// TIA Portal V15 export
// export: Created 2019-02-11T17:35:24.3452178Z, ExportSetting WithDefaults, WithReadOnly, DisplayName Totally Integrated Automation Portal, DisplayVersion V15 Update 2, DisplayName TIA Portal Openness, DisplayVersion V15 Update 2, DisplayName STEP 7 Professional, DisplayVersion V15 Update 2, DisplayName STEP 7 Safety, DisplayVersion V15, DisplayName WinCC Professional, DisplayVersion V15 Update 2, DisplayName SIMATIC Visualization Architect, DisplayVersion V15 Update 1
DATA_BLOCK "FGDB_ROBNAME@StudWeld"   // DB37
{ S7_Optimized_Access := 'FALSE' }
AUTHOR : integra
FAMILY : SUB
VERSION : 1.0
// stored: AutoNumber true, CodeModifiedDate 2019-02-11T17:32:35.5704024Z, CompileDate 2019-02-11T17:35:11.3679114Z, CreationDate 2019-02-11T17:32:35.4877706Z, DBAccessibleFromOPCUA true, InstanceOfName iSF_TECH_ROBOT_STUD_WELDING, InstanceOfNumber 15, InstanceOfType FB, InterfaceModifiedDate 2019-02-11T17:15:28.4108745Z, IsConsistent true, IsKnowHowProtected false, ModifiedDate 2019-02-11T17:32:35.5704024Z, ParameterModified 2018-10-24T10:12:24.9668345Z, StructureModified 2018-10-24T10:12:24.9668345Z, UDAEnableTagReadback false
"iSF_TECH_ROBOT_STUD_WELDING"
   // VAR_INPUT
   //    fct : Int;
   //    safetyStop : Bool;
   //    functionPoint : String[6];
   //    identType : String[12];
   //    releaseALUwelding : Bool;
   // END_VAR
   // VAR_OUTPUT
   //    qualityDataSent : Bool;
   //    qStop : Bool;
   //    counterParts : Int;
   //    counterNIOpoints : Int;
   //    counterIOpoints : Int;
   //    requestALUwelding : Bool;
   //    headClean1HomePosition : Bool;
   //    headClean2HomePosition : Bool;
   //    headClean3HomePosition : Bool;
   //    fault : Bool;
   // END_VAR
   // VAR_IN_OUT
   //    IfcFGExternal : "iUDT_IFC_SYS_EXTERNAL_ALARM";
   //    IfcTECH : "iUDT_IFC_ROBOT_TECH";
   //    IfcAcyclicdata : "iUDT_IFC_ROBOT_ACYCLICDATA";
   //    ident : Variant;
   //    IfcTLG : "iUDT_IFC_TLG";
   //    TLG_MQDV : "iUDT_TLG_MQDV_ROBOT";
   //    TLG_ENEV : "iUDT_TLG_ENEV";
   //    In_PI_TECH : "iUDT_PI_ROBOT_ADRxx48_TECH";
   //    Out_PO_TECH : "iUDT_PO_ROBOT_ADRxx48_TECH";
   // END_VAR
   // VAR
   //    F : Struct
   //       wrongID : Bool;
   //       notReady : Bool;
   //       boltControllerfault : Bool;
   //       plus : Bool;
   //       pointsNIO : Bool;
   //       partsNIO : Bool;
   //    END_STRUCT;
   //    Masks : Struct
   //       disableFault1_8 : Byte;
   //       prodRelevantFault1_8 : Byte;
   //    END_STRUCT;
   //    LastState : Struct
   //       fault1_8 : Byte;
   //    END_STRUCT;
   //    Tmr : Struct
   //       s1 { S7_SetPoint := 'True'} : Int;
   //       a1 : Int;
   //    END_STRUCT;
   //    TmrB : Struct
   //       "1_EnableDelayTime" : Bool;
   //       "1_RunDelayTime" : Bool;
   //       "1_DoneDelayTime" : Bool;
   //    END_STRUCT;
   //    D : Struct
   //       visuAck : Bool;
   //       evaluatedNIOCounter : Bool;
   //    END_STRUCT;
   //    V : Struct
   //       pointsNIO : Struct
   //          actual : Int;
   //          limitValue { S7_SetPoint := 'True'} : Int;
   //       END_STRUCT;
   //       partsNIO : Struct
   //          actual : Int;
   //          limitValue { S7_SetPoint := 'True'} : Int;
   //          resetCounter { S7_SetPoint := 'True'} : Int;
   //          actualCounter : Int;
   //       END_STRUCT;
   //       plusNIO : Struct
   //          actual : Int;
   //          limitValue { S7_SetPoint := 'True'} : Int;
   //          resetCounter { S7_SetPoint := 'True'} : Int;
   //          actualCounter : Int;
   //       END_STRUCT;
   //    END_STRUCT;
   //    TECH : Struct
   //       ID : Byte;
   //       ready : Bool;
   //       noFault : Bool;
   //       warning : Bool;
   //       noEstop : Bool;
   //       noUserProtection : Bool;
   //       plus : Bool;
   //       tolerance : Bool;
   //       requestALUwelding : Bool;
   //       preWarningHeadClean : Bool;
   //       requestHeadClean : Bool;
   //       headCleanOverflow : Bool;
   //       headCleanRotateSwitch : Bool;
   //       headClean1WorkPosition : Bool;
   //       headClean1HomePosition : Bool;
   //       headClean2WorkPosition : Bool;
   //       headClean2HomePosition : Bool;
   //       headClean3WorkPosition : Bool;
   //       headClean3HomePosition : Bool;
   //       technoBit19 : Bool;
   //       technoBit20 : Bool;
   //       technoBit21 : Bool;
   //       technoBit22 : Bool;
   //       technoBit23 : Bool;
   //       technoBit24 : Bool;
   //       technoBit25 : Bool;
   //       technoBit26 : Bool;
   //       technoBit27 : Bool;
   //       technoBit28 : Bool;
   //       technoBit29 : Bool;
   //       technoBit30 : Bool;
   //       technoBit31 : Bool;
   //       technoBit32 : Bool;
   //       technoBit33 : Bool;
   //       technoBit34 : Bool;
   //       technoBit35 : Bool;
   //       technoBit36 : Bool;
   //       technoBit37 : Bool;
   //       technoBit38 : Bool;
   //       technoBit39 : Bool;
   //       technoBit40 : Bool;
   //    END_STRUCT;
   //    TECH_OUT : Struct
   //       ID { ExternalWritable := 'False'} : Byte;
   //       releaseALUwelding : Bool;
   //       technoBit2 : Bool;
   //       technoBit3 : Bool;
   //       technoBit4 : Bool;
   //       technoBit5 : Bool;
   //       technoBit6 : Bool;
   //       technoBit7 : Bool;
   //       technoBit8 : Bool;
   //       technoBit9 : Bool;
   //       technoBit10 : Bool;
   //       technoBit11 : Bool;
   //       technoBit12 : Bool;
   //       technoBit13 : Bool;
   //       technoBit14 : Bool;
   //       technoBit15 : Bool;
   //       technoBit16 : Bool;
   //       technoBit17 : Bool;
   //       technoBit18 : Bool;
   //       technoBit19 : Bool;
   //       technoBit20 : Bool;
   //       technoBit21 : Bool;
   //       technoBit22 : Bool;
   //       technoBit23 : Bool;
   //       technoBit24 : Bool;
   //       technoBit25 : Bool;
   //       technoBit26 : Bool;
   //       technoBit27 : Bool;
   //       technoBit28 : Bool;
   //       technoBit29 : Bool;
   //       technoBit30 : Bool;
   //       technoBit31 : Bool;
   //       technoBit32 : Bool;
   //       technoBit33 : Bool;
   //       technoBit34 : Bool;
   //       technoBit35 : Bool;
   //       technoBit36 : Bool;
   //       technoBit37 : Bool;
   //       technoBit38 : Bool;
   //       technoBit39 : Bool;
   //       technoBit40 : Bool;
   //    END_STRUCT;
   //    PLUS : "iIF_ROBOT_PLUS";
   // END_VAR
BEGIN
END_DATA_BLOCK
